TYPE ST_LeicaFeedback :
STRUCT
	pos: ARRAY[0..2] OF LREAL;
	quat: ARRAY[0..3] OF LREAL;
END_STRUCT
END_TYPE

(* stored: Version 1.1.0.1, ProductVersion 3.1.4022.7
   DUT ST_LeicaFeedback: Id {8f910718-ad9e-498f-85d0-3eef97266d8e} *)
